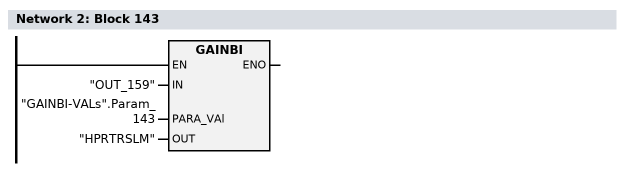
NETWORK
TITLE = Block 143
      CALL  "GAINBI" (
           IN                       := "OUT_159",
           PARA_VAl                 := "GAINBI-VALs".Param_143,
           OUT                      := "HPRTRSLM");
      NOP   0;
END_FUNCTION

FUNCTION "Sheet 23 (RSM)" : VOID	// FC 62
TITLE = Sheet 23 (RSM)
//HP ROTOR STRESS LIMIT (Digital)
AUTHOR : RJ
FAMILY : RSM
VERSION : 0.1
BEGIN
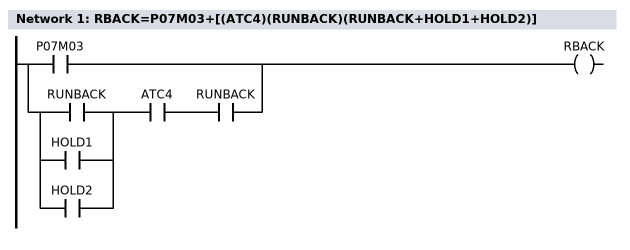
NETWORK
TITLE = RBACK=P07M03+[(ATC4)(RUNBACK)(RUNBACK+HOLD1+HOLD2)]
      O     "P07M03";
      O;
      A(;
      O     "RUNBACK";
      O     "HOLD1";
      O     "HOLD2";
      );
      A     "ATC4";
      A     "RUNBACK";
      =     "RBACK";
NETWORK
TITLE = P01M02=[FF(HILDPB,[NORLDPB+~BR+LDEQDMD])][DVTRUE]
      A(;
      A     "HILDPB";
      S     "HILDRAT";
      A(;
      O     "NORLDPB";
      ON    "BR";
      O     "LDEQDMD";
      );
      R     "HILDRAT";
      A     "HILDRAT";
      );
      A     "Constants_RSM".DVTRUE;
      =     "P01M02";
END_FUNCTION

FUNCTION "Sheet 24 (RSM)" : VOID	// FC 63
TITLE = Sheet 24 (RSM)
//ATC TARGET (Analog)
AUTHOR : RJ
FAMILY : RSM
VERSION : 0.1
BEGIN
NETWORK
TITLE = Blocks X712, X715
      A     "RES1";
      =     L 0.0;
      BLD   103;
      A(;
      A     "HLD1";
      =     L 0.1;
      BLD   103;
      CALL  "XTRANSF" (
           PV_Y                     := "REFDMD",
           CAS_N                    := "OUT_X171",
           FLAG                     := L 0.1,
           PARA_VAl                 := "XTRANSF_VALs".Param_X712,
           OUTPUT                   := "OUT_X712");
      A     BR;
      );
      JNB   _001;
      CALL  "XTRANSF" (
           PV_Y                     := "REFF1",
           CAS_N                    := "OUT_X712",
           FLAG                     := L 0.0,
           PARA_VAl                 := "XTRANSF_VALs".Param_X715,
           OUTPUT                   := "OUT_X715");
_001: NOP   0;
NETWORK
TITLE = Blocks X717, X721
      A     "RES3";
      =     L 0.0;
      BLD   103;
      A(;
      A     "RES2";
      =     L 0.1;
      BLD   103;
      CALL  "XTRANSF" (
           PV_Y                     := "REFF2",
           CAS_N                    := "OUT_X715",
           FLAG                     := L 0.1,
           PARA_VAl                 := "XTRANSF_VALs".Param_X717,
           OUTPUT                   := "DMDTEMP2");
      A     BR;
      );
      JNB   _002;
      CALL  "XTRANSF" (
           PV_Y                     := "REFF3",
           CAS_N                    := "DMDTEMP2",
           FLAG                     := L 0.0,
           PARA_VAl                 := "XTRANSF_VALs".Param_X721,
           OUTPUT                   := "OUT_X721");
_002: NOP   0;
NETWORK
TITLE = Blocks X723, X725
      A     "RES5";
      =     L 0.0;
      BLD   103;
      A(;
      A     "RES4";
      =     L 0.1;
      BLD   103;
      CALL  "XTRANSF" (
           PV_Y                     := "REFF4",
           CAS_N                    := "OUT_X721",
           FLAG                     := L 0.1,
           PARA_VAl                 := "XTRANSF_VALs".Param_X723,
           OUTPUT                   := "OUT_X723");
      A     BR;
      );
      JNB   _003;
      CALL  "XTRANSF" (
           PV_Y                     := "REFF5",
           CAS_N                    := "DMDTEMP3",
           FLAG                     := L 0.0,
           PARA_VAl                 := "XTRANSF_VALs".Param_X725,
           OUTPUT                   := "DMDTEMP3");
_003: NOP   0;
NETWORK
TITLE = Blocks X741, X743
      A     "RBACK";
      =     L 0.0;
      BLD   103;
      A(;
      A     "EXC1";
      =     L 0.1;
      BLD   103;
      CALL  "XTRANSF" (
           PV_Y                     := "Constants_RSM".A40,
           CAS_N                    := "DMDTEMP3",
           FLAG                     := L 0.1,
           PARA_VAl                 := "XTRANSF_VALs".Param_X741,
           OUTPUT                   := "OUT_X741");
      A     BR;
      );
      JNB   _004;
      CALL  "XTRANSF" (
           PV_Y                     := "ATCSPDRF",
           CAS_N                    := "OUT_X741",
           FLAG                     := L 0.0,
           PARA_VAl                 := "XTRANSF_VALs".Param_X743,
           OUTPUT                   := "DEHDMD");
_004: NOP   0;
NETWORK
TITLE = Blocks X701, X707
      A     "DEHDMD1";
      =     L 0.0;
      BLD   103;
      A(;
      A     "P15M13";
      =     L 0.1;
      BLD   103;
      CALL  "XTRANSF" (
           PV_Y                     := "Constants_RSM".A40,
           CAS_N                    := "DEHDMD",
           FLAG                     := L 0.1,
           PARA_VAl                 := "XTRANSF_VALs".Param_X701,
           OUTPUT                   := "OUT_X701");
      A     BR;
      );
      JNB   _005;
      CALL  "XTRANSF" (
           PV_Y                     := "Constants_RSM".A40,
           CAS_N                    := "OUT_X701",
           FLAG                     := L 0.0,
           PARA_VAl                 := "XTRANSF_VALs".Param_X707,
           OUTPUT                   := "OUT_X707");
_005: NOP   0;
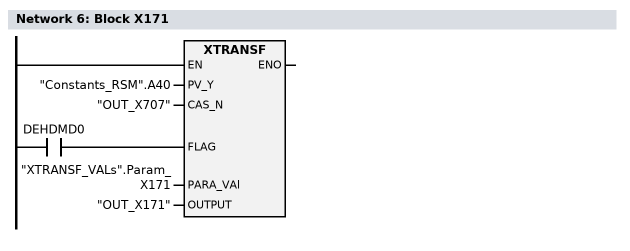
NETWORK
TITLE = Block X171
      A     "DEHDMD0";
      =     L 0.0;
      BLD   103;
      CALL  "XTRANSF" (
           PV_Y                     := "Constants_RSM".A40,
           CAS_N                    := "OUT_X707",
           FLAG                     := L 0.0,
           PARA_VAl                 := "XTRANSF_VALs".Param_X171,
           OUTPUT                   := "OUT_X171");
      NOP   0;
END_FUNCTION

FUNCTION "Sheet 25 (RSM)" : VOID	// FC 64
TITLE = Sheet 25 (RSM)
//TRANSFER DELAY (Digital)
AUTHOR : RJ
FAMILY : RSM
VERSION : 0.1
BEGIN
NETWORK
TITLE = CRSBO4=FF[(AFLAG)(ATC4),(ATC4)(Z871)]
//Z871=ON(CRSBO4)
      A(;
      A     "AFLAG";
      A     "ATC4";
      S     "CRSBO4";
      A     "Z871";
      A     "ATC4";
      R     "CRSBO4";
      A     "CRSBO4";
      );
      =     "CRSBO4";
      A     "CRSBO4";
      L     "RSMTime_VALs".T1ON;
      SD    T 1;
      NOP   0;
      NOP   0;
      NOP   0;
      A     T 1;
      =     "Z871";
END_FUNCTION

FUNCTION "Sheet 26 (RSM)" : VOID	// FC 65
TITLE = Sheet 26 (RSM)
//LADDERS 35, 128, RESONANCE RANGE LOGIC (Digital)
AUTHOR : RJ
FAMILY : RSM
VERSION : 0.1
BEGIN
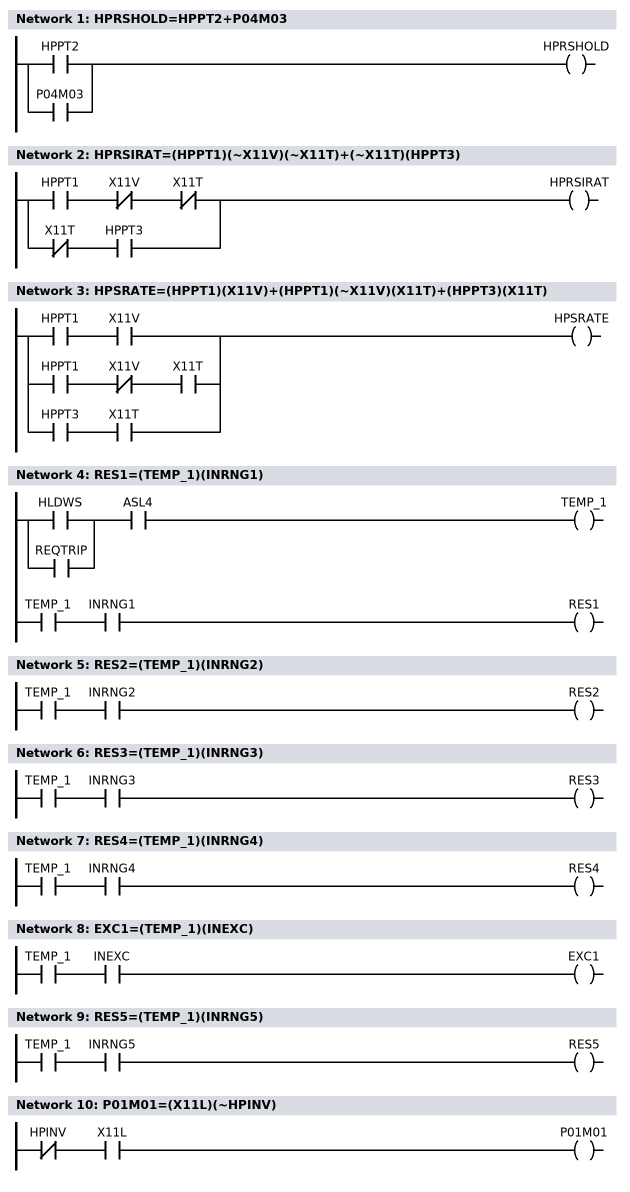
NETWORK
TITLE = HPRSHOLD=HPPT2+P04M03
      O     "HPPT2";
      O     "P04M03";
      =     "HPRSHOLD";
NETWORK
TITLE = HPRSIRAT=(HPPT1)(~X11V)(~X11T)+(~X11T)(HPPT3)
      A     "HPPT1";
      AN    "X11V";
      AN    "X11T";
      O;
      AN    "X11T";
      A     "HPPT3";
      =     "HPRSIRAT";
NETWORK
TITLE = HPSRATE=(HPPT1)(X11V)+(HPPT1)(~X11V)(X11T)+(HPPT3)(X11T)
      A     "HPPT1";
      A     "X11V";
      O;
      A     "HPPT1";
      AN    "X11V";
      A     "X11T";
      O;
      A     "HPPT3";
      A     "X11T";
      =     "HPSRATE";
NETWORK
TITLE = RES1=(TEMP_1)(INRNG1)
//TEMP_1=(ASL4)(HLDWS+REQTRIP)
      A(;
      O     "HLDWS";
      O     "REQTRIP";
      );
      A     "ASL4";
      =     "TEMP_1";
      A     "TEMP_1";
      A     "INRNG1";
      =     "RES1";
NETWORK
TITLE = RES2=(TEMP_1)(INRNG2)
      A     "TEMP_1";
      A     "INRNG2";
      =     "RES2";
NETWORK
TITLE = RES3=(TEMP_1)(INRNG3)
      A     "TEMP_1";
      A     "INRNG3";
      =     "RES3";
NETWORK
TITLE = RES4=(TEMP_1)(INRNG4)
      A     "TEMP_1";
      A     "INRNG4";
      =     "RES4";
NETWORK
TITLE = EXC1=(TEMP_1)(INEXC)
      A     "TEMP_1";
      A     "INEXC";
      =     "EXC1";
NETWORK
TITLE = RES5=(TEMP_1)(INRNG5)
      A     "TEMP_1";
      A     "INRNG5";
      =     "RES5";
NETWORK
TITLE = P01M01=(X11L)(~HPINV)
      AN    "HPINV";
      A     "X11L";
      =     "P01M01";
END_FUNCTION

FUNCTION "Sheet 28 (RSM)" : VOID	// FC 66
TITLE = Sheet 28 (RSM)
//LADDERS 22, 500, 600, DIGITAL POINTERS TMAX & TWC LOGIC (Digital)
AUTHOR : RJ
FAMILY : RSM
VERSION : 0.1
BEGIN
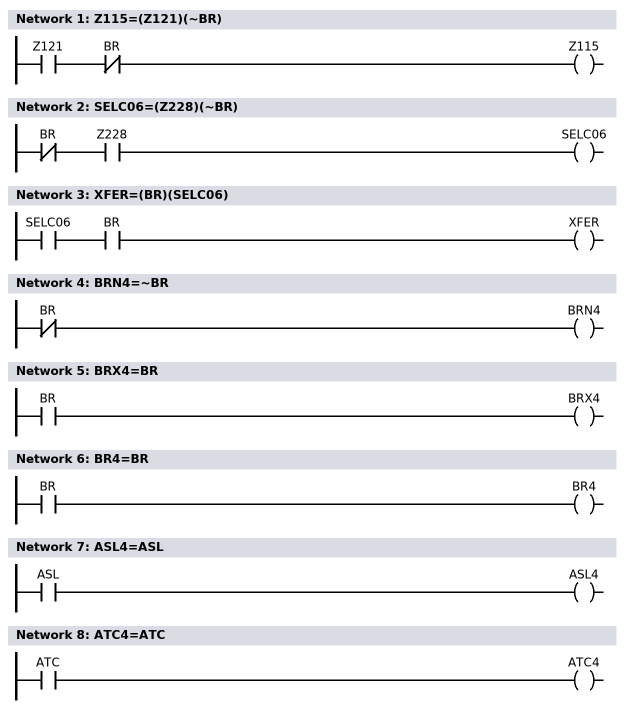
NETWORK
TITLE = Z115=(Z121)(~BR)
      A     "Z121";
      AN    "BR";
      =     "Z115";
NETWORK
TITLE = SELC06=(Z228)(~BR)
      AN    "BR";
      A     "Z228";
      =     "SELC06";
NETWORK
TITLE = XFER=(BR)(SELC06)
      A     "SELC06";
      A     "BR";
      =     "XFER";
NETWORK
TITLE = BRN4=~BR
      AN    "BR";
      =     "BRN4";
NETWORK
TITLE = BRX4=BR
      A     "BR";
      =     "BRX4";
NETWORK
TITLE = BR4=BR
      A     "BR";
      =     "BR4";
NETWORK
TITLE = ASL4=ASL
      A     "ASL";
      =     "ASL4";
NETWORK
TITLE = ATC4=ATC
      A     "ATC";
      =     "ATC4";
END_FUNCTION

FUNCTION "Sheet 29 (RSM)" : VOID	// FC 67
TITLE = Sheet 29 (RSM)
//LADDERS 29, 31, 500, FIRST STAGE STM > 75 *C (Digital)
AUTHOR : RJ
FAMILY : RSM
VERSION : 0.1
BEGIN
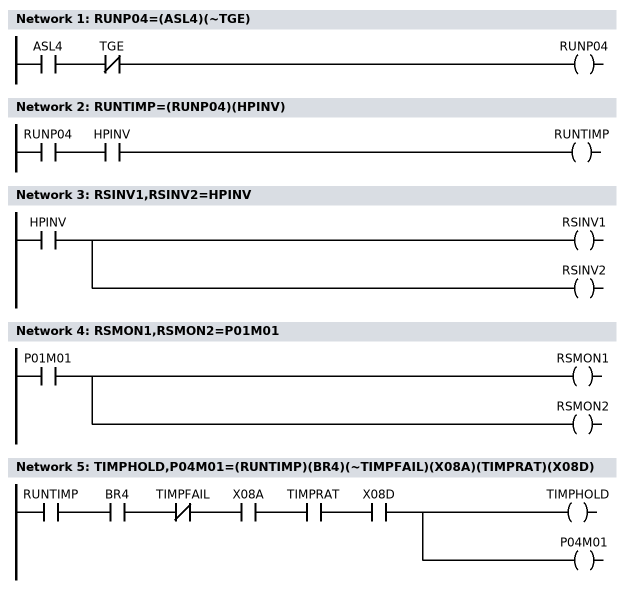
NETWORK
TITLE = RUNP04=(ASL4)(~TGE)
      A     "ASL4";
      AN    "TGE";
      =     "RUNP04";
NETWORK
TITLE = RUNTIMP=(RUNP04)(HPINV)
      A     "RUNP04";
      A     "HPINV";
      =     "RUNTIMP";
NETWORK
TITLE = RSINV1,RSINV2=HPINV
      A     "HPINV";
      =     "RSINV1";
      =     "RSINV2";
NETWORK
TITLE = RSMON1,RSMON2=P01M01
      A     "P01M01";
      =     "RSMON1";
      =     "RSMON2";
NETWORK
TITLE = TIMPHOLD,P04M01=(RUNTIMP)(BR4)(~TIMPFAIL)(X08A)(TIMPRAT)(X08D)
      A     "RUNTIMP";
      A     "BR4";
      AN    "TIMPFAIL";
      A     "X08A";
      A     "TIMPRAT";
      A     "X08D";
      =     "TIMPHOLD";
      =     "P04M01";
END_FUNCTION

FUNCTION "Sheet 27 (RSM)" : VOID	// FC 68
TITLE = Sheet 27 (RSM)
//LADDERS 43, 129, RTSHOLD (Digital)
AUTHOR : RJ
FAMILY : RSM
VERSION : 0.1
BEGIN
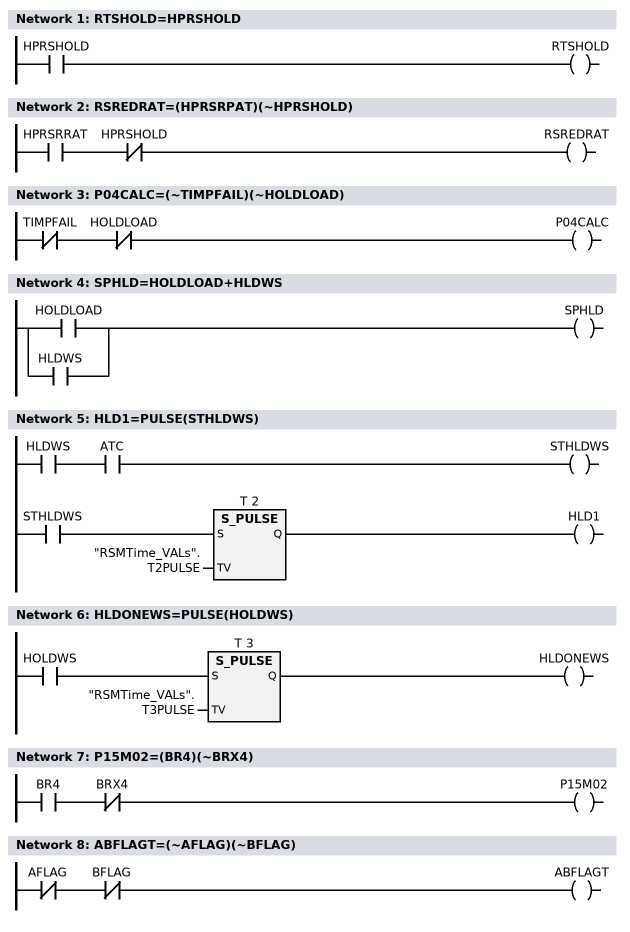
NETWORK
TITLE = RTSHOLD=HPRSHOLD
      A     "HPRSHOLD";
      =     "RTSHOLD";
NETWORK
TITLE = RSREDRAT=(HPRSRPAT)(~HPRSHOLD)
      A     "HPRSRRAT";
      AN    "HPRSHOLD";
      =     "RSREDRAT";
NETWORK
TITLE = P04CALC=(~TIMPFAIL)(~HOLDLOAD)
      AN    "TIMPFAIL";
      AN    "HOLDLOAD";
      =     "P04CALC";
NETWORK
TITLE = SPHLD=HOLDLOAD+HLDWS
      O     "HOLDLOAD";
      O     "HLDWS";
      =     "SPHLD";
NETWORK
TITLE = HLD1=PULSE(STHLDWS)
//STHLDWS=(HLDWS)(ATC)
      A     "HLDWS";
      A     "ATC";
      =     "STHLDWS";
      A     "STHLDWS";
      L     "RSMTime_VALs".T2PULSE;
      SP    T 2;
      NOP   0;
      NOP   0;
      NOP   0;
      A     T 2;
      =     "HLD1";
NETWORK
TITLE = HLDONEWS=PULSE(HOLDWS)
      A     "HOLDWS";
      L     "RSMTime_VALs".T3PULSE;
      SP    T 3;
      NOP   0;
      NOP   0;
      NOP   0;
      A     T 3;
      =     "HLDONEWS";
NETWORK
TITLE = P15M02=(BR4)(~BRX4)
      A     "BR4";
      AN    "BRX4";
      =     "P15M02";
NETWORK
TITLE = ABFLAGT=(~AFLAG)(~BFLAG)
      AN    "AFLAG";
      AN    "BFLAG";
      =     "ABFLAGT";
END_FUNCTION

FUNCTION "Sheet 30 (RSM)" : VOID	// FC 69
TITLE = Sheet 30 (RSM)
//LADDER 126, SYNC LOGIC & OVERRIDE (Digital)
AUTHOR : RJ
FAMILY : RSM
VERSION : 0.1
BEGIN
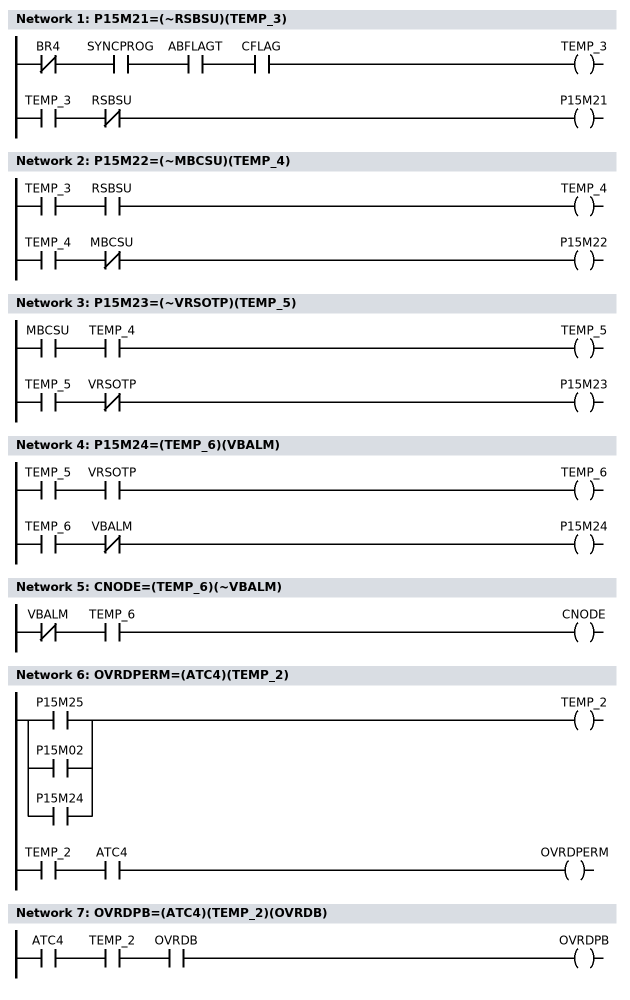
NETWORK
TITLE = P15M21=(~RSBSU)(TEMP_3)
//TEMP_3=(~BR4)(SYNCPROG)(ABFLAGT)(CFLAG)
      AN    "BR4";
      A     "SYNCPROG";
      A     "ABFLAGT";
      A     "CFLAG";
      =     "TEMP_3";
      A     "TEMP_3";
      AN    "RSBSU";
      =     "P15M21";
NETWORK
TITLE = P15M22=(~MBCSU)(TEMP_4)
//TEMP_4=(TEMP_3)(RSBSU)
      A     "TEMP_3";
      A     "RSBSU";
      =     "TEMP_4";
      A     "TEMP_4";
      AN    "MBCSU";
      =     "P15M22";
NETWORK
TITLE = P15M23=(~VRSOTP)(TEMP_5)
//TEMP_5=(MBCSU)(TEMP_4)
      A     "MBCSU";
      A     "TEMP_4";
      =     "TEMP_5";
      A     "TEMP_5";
      AN    "VRSOTP";
      =     "P15M23";
NETWORK
TITLE = P15M24=(TEMP_6)(VBALM)
//TEMP_6=(TEMP_5)(VRSOTP)
      A     "TEMP_5";
      A     "VRSOTP";
      =     "TEMP_6";
      A     "TEMP_6";
      AN    "VBALM";
      =     "P15M24";
NETWORK
TITLE = CNODE=(TEMP_6)(~VBALM)
      AN    "VBALM";
      A     "TEMP_6";
      =     "CNODE";
NETWORK
TITLE = OVRDPERM=(ATC4)(TEMP_2)
//TEMP_2=P15M25+P15M06+P15M24
      A(;
      O     "P15M25";
      O     "P15M02";
      O     "P15M24";
      );
      =     "TEMP_2";
      A     "TEMP_2";
      A     "ATC4";
      =     "OVRDPERM";
NETWORK
TITLE = OVRDPB=(ATC4)(TEMP_2)(OVRDB)
      A     "ATC4";
      A     "TEMP_2";
      A     "OVRDB";
      =     "OVRDPB";
END_FUNCTION

FUNCTION "Sheet 31 (RSM)" : VOID	// FC 70
TITLE = Sheet 31 (RSM)
//LADDER 33, ANTIC HP STRESS > LIMIT (Digital)
AUTHOR : RJ
FAMILY : RSM
VERSION : 0.1
BEGIN
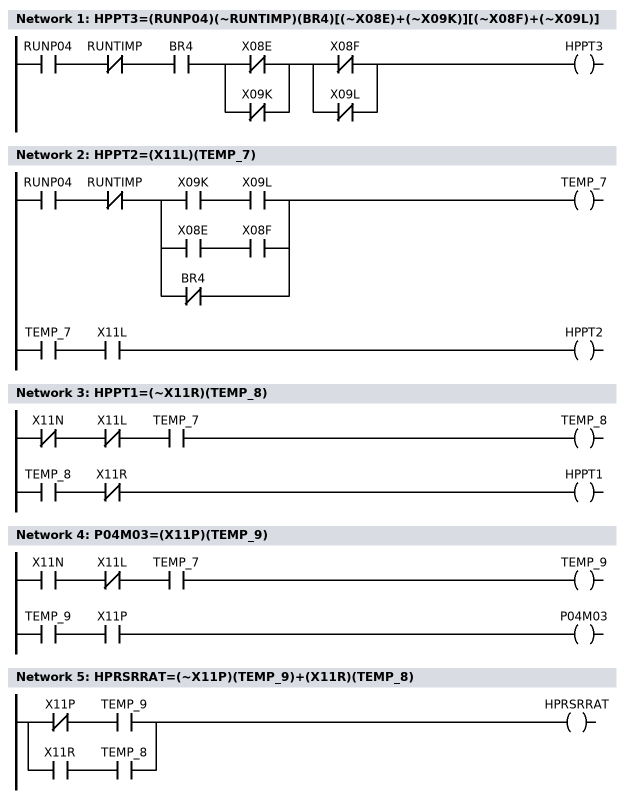
NETWORK
TITLE = HPPT3=(RUNP04)(~RUNTIMP)(BR4)[(~X08E)+(~X09K)][(~X08F)+(~X09L)]
      A     "RUNP04";
      AN    "RUNTIMP";
      A     "BR4";
      A(;
      ON    "X08E";
      ON    "X09K";
      );
      A(;
      ON    "X08F";
      ON    "X09L";
      );
      =     "HPPT3";
NETWORK
TITLE = HPPT2=(X11L)(TEMP_7)
//TEMP_7=(RUNP04)(~RUNTIMP)[(X09K)(X09L)+(X08E)(X08F)+(~BR4)]
      A     "RUNP04";
      AN    "RUNTIMP";
      A(;
      A     "X09K";
      A     "X09L";
      O;
      A     "X08E";
      A     "X08F";
      ON    "BR4";
      );
      =     "TEMP_7";
      A     "TEMP_7";
      A     "X11L";
      =     "HPPT2";
NETWORK
TITLE = HPPT1=(~X11R)(TEMP_8)
//TEMP_8=(~X11N)(~X11L)(TEMP_7)
      AN    "X11N";
      AN    "X11L";
      A     "TEMP_7";
      =     "TEMP_8";
      A     "TEMP_8";
      AN    "X11R";
      =     "HPPT1";
NETWORK
TITLE = P04M03=(X11P)(TEMP_9)
//TEMP_9=(X11N)(~X11L)(TEMP_7)
      A     "X11N";
      AN    "X11L";
      A     "TEMP_7";
      =     "TEMP_9";
      A     "TEMP_9";
      A     "X11P";
      =     "P04M03";
NETWORK
TITLE = HPRSRRAT=(~X11P)(TEMP_9)+(X11R)(TEMP_8)
      AN    "X11P";
      A     "TEMP_9";
      O;
      A     "X11R";
      A     "TEMP_8";
      =     "HPRSRRAT";
END_FUNCTION

FUNCTION "Sheet 32 (RSM)" : VOID	// FC 71
TITLE = Sheet 32 (RSM)
//LADDERS 37, 125, 130, SYNC LOGIC & OVERRIDE (Digital)
AUTHOR : RJ
FAMILY : RSM
VERSION : 0.1
BEGIN
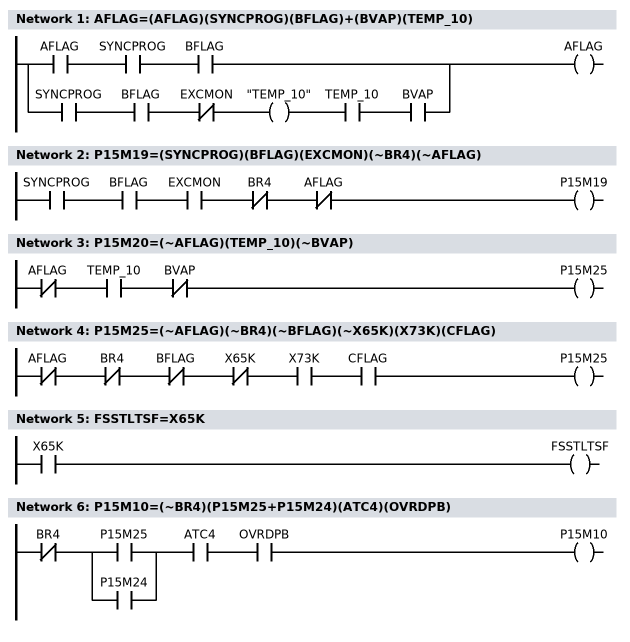
NETWORK
TITLE = AFLAG=(AFLAG)(SYNCPROG)(BFLAG)+(BVAP)(TEMP_10)
//TEMP_10=(SYNCPROG)(BFLAG)(~EXCMON)
      A     "AFLAG";
      A     "SYNCPROG";
      A     "BFLAG";
      O(;
      A     "SYNCPROG";
      A     "BFLAG";
      AN    "EXCMON";
      =     "TEMP_10";
      A     "TEMP_10";
      A     "BVAP";
      );
      =     "AFLAG";
NETWORK
TITLE = P15M19=(SYNCPROG)(BFLAG)(EXCMON)(~BR4)(~AFLAG)
      A     "SYNCPROG";
      A     "BFLAG";
      A     "EXCMON";
      AN    "BR4";
      AN    "AFLAG";
      =     "P15M19";
NETWORK
TITLE = P15M20=(~AFLAG)(TEMP_10)(~BVAP)
      AN    "AFLAG";
      A     "TEMP_10";
      AN    "BVAP";
      =     "P15M25";
NETWORK
TITLE = P15M25=(~AFLAG)(~BR4)(~BFLAG)(~X65K)(X73K)(CFLAG)
      AN    "AFLAG";
      AN    "BR4";
      AN    "BFLAG";
      AN    "X65K";
      A     "X73K";
      A     "CFLAG";
      =     "P15M25";
NETWORK
TITLE = FSSTLTSF=X65K
      A     "X65K";
      =     "FSSTLTSF";
NETWORK
TITLE = P15M10=(~BR4)(P15M25+P15M24)(ATC4)(OVRDPB)
      AN    "BR4";
      A(;
      O     "P15M25";
      O     "P15M24";
      );
      A     "ATC4";
      A     "OVRDPB";
      =     "P15M10";
END_FUNCTION

FUNCTION "Sheet 33 (RSM)" : VOID	// FC 72
TITLE = Sheet 33 (RSM)
//LADDER 124, 127, SYNC LOGIC & TVGVINIT (Digital)
AUTHOR : RJ
FAMILY : RSM
VERSION : 0.1
BEGIN
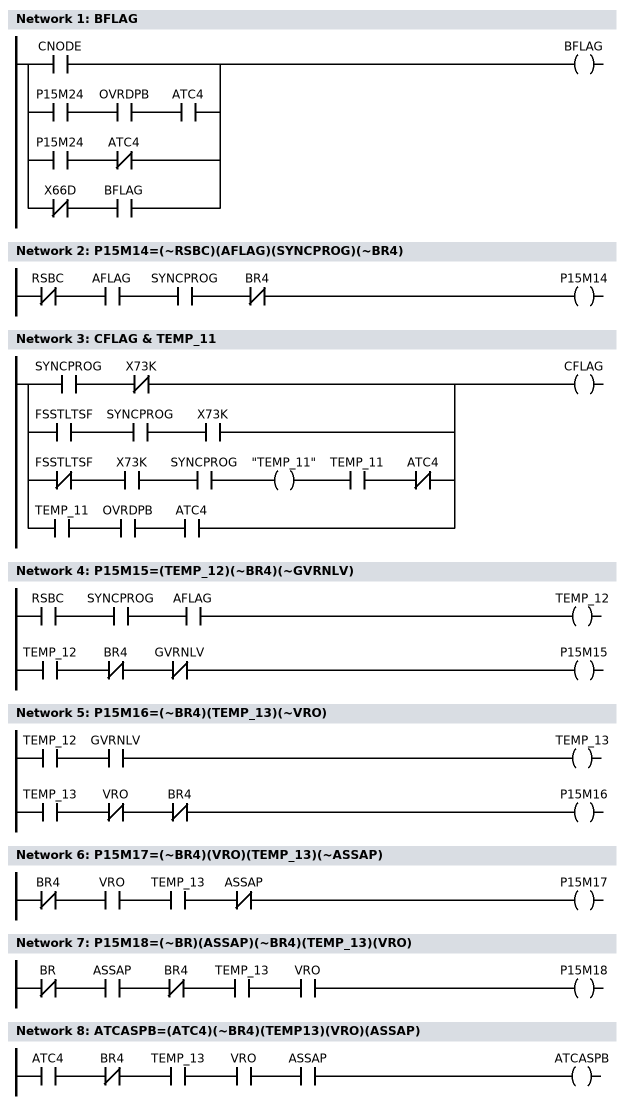
NETWORK
TITLE = BFLAG
//BFLAG=CNODE+(P15M24)(OVRDPB)(ATC4)+(P15M24)(~ATC4)+(~X66D)(BFLAG)
      O     "CNODE";
      O;
      A     "P15M24";
      A     "OVRDPB";
      A     "ATC4";
      O;
      A     "P15M24";
      AN    "ATC4";
      O;
      AN    "X66D";
      A     "BFLAG";
      =     "BFLAG";
NETWORK
TITLE = P15M14=(~RSBC)(AFLAG)(SYNCPROG)(~BR4)
      AN    "RSBC";
      A     "AFLAG";
      A     "SYNCPROG";
      AN    "BR4";
      =     "P15M14";
NETWORK
TITLE = CFLAG & TEMP_11
//CFLAG=(SYNCPROG)(~X73K)+(FSSTLTSF)(SYNCPROG)(X73K)+(~ATC4)(TEMP_11)+(TEMP_11)
//(OVRDPB)(ATC4)
//
//TEMP_11=(~FSSTLTSF)(X73K)(SYNCPROG)
//
      A     "SYNCPROG";
      AN    "X73K";
      O(;
      A     "FSSTLTSF";
      A     "SYNCPROG";
      A     "X73K";
      );
      O(;
      AN    "FSSTLTSF";
      A     "X73K";
      A     "SYNCPROG";
      =     "TEMP_11";
      A     "TEMP_11";
      AN    "ATC4";
      );
      O;
      A     "TEMP_11";
      A     "OVRDPB";
      A     "ATC4";
      =     "CFLAG";
NETWORK
TITLE = P15M15=(TEMP_12)(~BR4)(~GVRNLV)
//TEMP_12=(RSBC)(SYNCPROG)(AFLAG)
      A     "RSBC";
      A     "SYNCPROG";
      A     "AFLAG";
      =     "TEMP_12";
      A     "TEMP_12";
      AN    "BR4";
      AN    "GVRNLV";
      =     "P15M15";
NETWORK
TITLE = P15M16=(~BR4)(TEMP_13)(~VRO)
//TEMP_13=(TEMP_12)(GVRNLV)
      A     "TEMP_12";
      A     "GVRNLV";
      =     "TEMP_13";
      A     "TEMP_13";
      AN    "VRO";
      AN    "BR4";
      =     "P15M16";
NETWORK
TITLE = P15M17=(~BR4)(VRO)(TEMP_13)(~ASSAP)
      AN    "BR4";
      A     "VRO";
      A     "TEMP_13";
      AN    "ASSAP";
      =     "P15M17";
NETWORK
TITLE = P15M18=(~BR)(ASSAP)(~BR4)(TEMP_13)(VRO)
      AN    "BR";
      A     "ASSAP";
      AN    "BR4";
      A     "TEMP_13";
      A     "VRO";
      =     "P15M18";
NETWORK
TITLE = ATCASPB=(ATC4)(~BR4)(TEMP13)(VRO)(ASSAP)
      A     "ATC4";
      AN    "BR4";
      A     "TEMP_13";
      A     "VRO";
      A     "ASSAP";
      =     "ATCASPB";
END_FUNCTION

FUNCTION "Sheet 34 (RSM)" : VOID	// FC 73
TITLE = Sheet 34 (RSM)
//LADDERS 122, 123, 135, SET SPEED PLATEAU (Digital)
AUTHOR : RJ
FAMILY : RSM
VERSION : 0.1
BEGIN
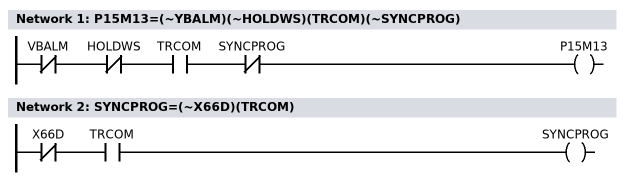
NETWORK
TITLE = P15M13=(~YBALM)(~HOLDWS)(TRCOM)(~SYNCPROG)
      AN    "VBALM";
      AN    "HOLDWS";
      A     "TRCOM";
      AN    "SYNCPROG";
      =     "P15M13";
NETWORK
TITLE = SYNCPROG=(~X66D)(TRCOM)
      AN    "X66D";
      A     "TRCOM";
      =     "SYNCPROG";
END_FUNCTION

FUNCTION "Sheet 35 (RSM)" : VOID	// FC 74
TITLE = Sheet 35 (RSM)
//LADDER 120, 121, P15 ALARMS ESTIMATE ROLL TIME LOGIC & ATC VPL (Digital)
AUTHOR : RJ
FAMILY : RSM
VERSION : 0.1
BEGIN
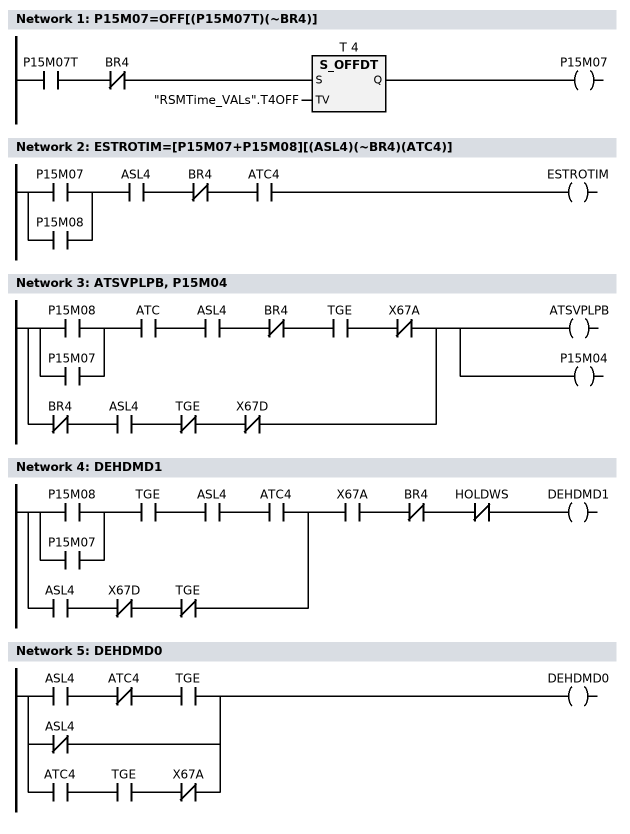
NETWORK
TITLE = P15M07=OFF[(P15M07T)(~BR4)]
      A     "P15M07T";
      AN    "BR4";
      L     "RSMTime_VALs".T4OFF;
      SF    T 4;
      NOP   0;
      NOP   0;
      NOP   0;
      A     T 4;
      =     "P15M07";
NETWORK
TITLE = ESTROTIM=[P15M07+P15M08][(ASL4)(~BR4)(ATC4)]
      A(;
      O     "P15M07";
      O     "P15M08";
      );
      A     "ASL4";
      AN    "BR4";
      A     "ATC4";
      =     "ESTROTIM";
NETWORK
TITLE = ATSVPLPB, P15M04
//ATSVPLPB,P15M04=[(P15M08+P15M07)(ATC)(ASL4)(~BR4)(TGE)(~X67A)]+[(~BR4)(ASL4)
//(~TGE)(~X67D)]
      A(;
      O     "P15M08";
      O     "P15M07";
      );
      A     "ATC";
      A     "ASL4";
      AN    "BR4";
      A     "TGE";
      AN    "X67A";
      O;
      AN    "BR4";
      A     "ASL4";
      AN    "TGE";
      AN    "X67D";
      =     "ATSVPLPB";
      =     "P15M04";
NETWORK
TITLE = DEHDMD1
//DEHDMD1=[{(P15M08+P15M07)(TGE)(ASL4)(ATC4)}+{(ASL4)(~X67D)(~TGE)}][X67A][~BR4]
//[~HOLDWS]
      A(;
      A(;
      O     "P15M08";
      O     "P15M07";
      );
      A     "TGE";
      A     "ASL4";
      A     "ATC4";
      O;
      A     "ASL4";
      AN    "X67D";
      AN    "TGE";
      );
      A     "X67A";
      AN    "BR4";
      AN    "HOLDWS";
      =     "DEHDMD1";
NETWORK
TITLE = DEHDMD0
//DEHDMD0=[(ASL4)(~ATC4)(TGE)]+[~ASL4]+[(ASL4)(TGE)(~X67A)]
      A     "ASL4";
      AN    "ATC4";
      A     "TGE";
      ON    "ASL4";
      O;
      A     "ATC4";
      A     "TGE";
      AN    "X67A";
      =     "DEHDMD0";
END_FUNCTION

FUNCTION "Sheet 36 (RSM)" : VOID	// FC 75
TITLE = Sheet 36 (RSM)
//LADDER 41, 119, P15 ALARMS (Digital)
AUTHOR : RJ
FAMILY : RSM
VERSION : 0.1
BEGIN
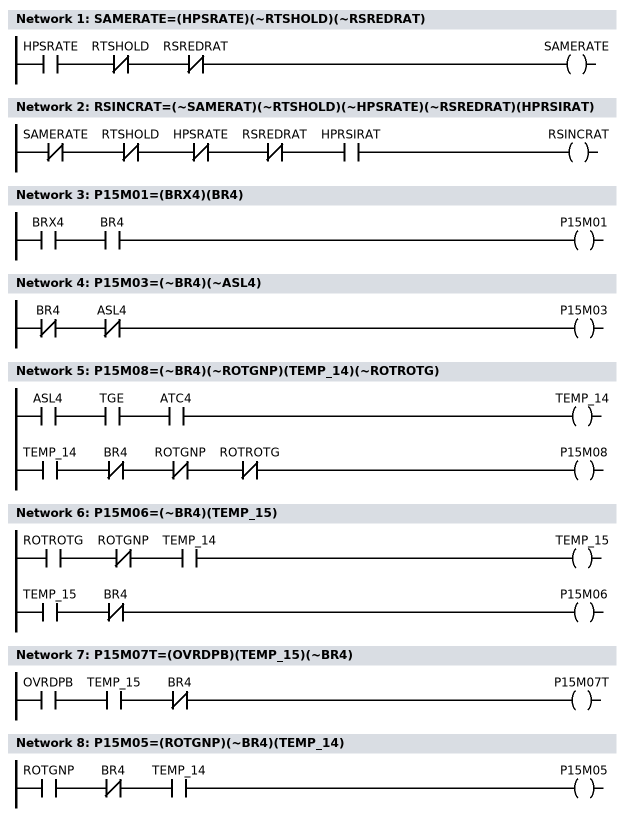
NETWORK
TITLE = SAMERATE=(HPSRATE)(~RTSHOLD)(~RSREDRAT)
      A     "HPSRATE";
      AN    "RTSHOLD";
      AN    "RSREDRAT";
      =     "SAMERATE";
NETWORK
TITLE = RSINCRAT=(~SAMERAT)(~RTSHOLD)(~HPSRATE)(~RSREDRAT)(HPRSIRAT)
      AN    "SAMERATE";
      AN    "RTSHOLD";
      AN    "HPSRATE";
      AN    "RSREDRAT";
      A     "HPRSIRAT";
      =     "RSINCRAT";
NETWORK
TITLE = P15M01=(BRX4)(BR4)
      A     "BRX4";
      A     "BR4";
      =     "P15M01";
NETWORK
TITLE = P15M03=(~BR4)(~ASL4)
      AN    "BR4";
      AN    "ASL4";
      =     "P15M03";
NETWORK
TITLE = P15M08=(~BR4)(~ROTGNP)(TEMP_14)(~ROTROTG)
//TEMP_14=(ASL4)(TGE)(ATC4)
      A     "ASL4";
      A     "TGE";
      A     "ATC4";
      =     "TEMP_14";
      A     "TEMP_14";
      AN    "BR4";
      AN    "ROTGNP";
      AN    "ROTROTG";
      =     "P15M08";
NETWORK
TITLE = P15M06=(~BR4)(TEMP_15)
//TEMP_15=(ROTROTG)(~ROTGNP)(TEMP_14)
      A     "ROTROTG";
      AN    "ROTGNP";
      A     "TEMP_14";
      =     "TEMP_15";
      A     "TEMP_15";
      AN    "BR4";
      =     "P15M06";
NETWORK
TITLE = P15M07T=(OVRDPB)(TEMP_15)(~BR4)
      A     "OVRDPB";
      A     "TEMP_15";
      AN    "BR4";
      =     "P15M07T";
NETWORK
TITLE = P15M05=(ROTGNP)(~BR4)(TEMP_14)
      A     "ROTGNP";
      AN    "BR4";
      A     "TEMP_14";
      =     "P15M05";
END_FUNCTION

FUNCTION "Sheet 37 (RSM)" : VOID	// FC 76
TITLE = Sheet 37 (RSM)
//GENERATOR AND EXCITOR TEMPERATURES (Analog)
AUTHOR : RJ
FAMILY : RSM
VERSION : 0.1
BEGIN
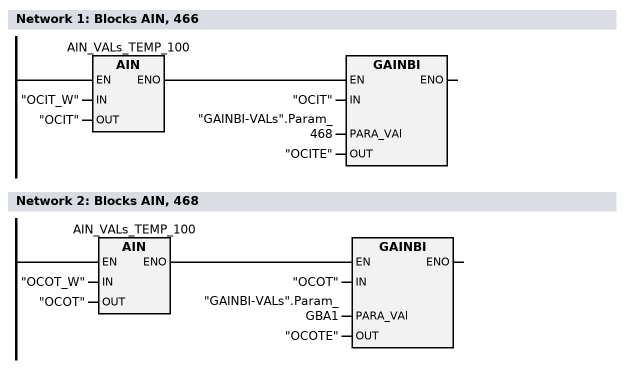
NETWORK
TITLE = Blocks AIN, 466
      A(;
      CALL  "AIN" , "AIN_VALs_TEMP_100" (
           IN                       := "OCIT_W",
           OUT                      := "OCIT");
      A     BR;
      );
      JNB   _001;
      CALL  "GAINBI" (
           IN                       := "OCIT",
           PARA_VAl                 := "GAINBI-VALs".Param_468,
           OUT                      := "OCITE");
_001: NOP   0;
NETWORK
TITLE = Blocks AIN, 468
      A(;
      CALL  "AIN" , "AIN_VALs_TEMP_100" (
           IN                       := "OCOT_W",
           OUT                      := "OCOT");
      A     BR;
      );
      JNB   _002;
      CALL  "GAINBI" (
           IN                       := "OCOT",
           PARA_VAl                 := "GAINBI-VALs".Param_GBA1,
           OUT                      := "OCOTE");
_002: NOP   0;
END_FUNCTION

FUNCTION "Sheet 2 (ATC)" : VOID	// FC 77
TITLE = Sheet 2 (ATC)
//LADDER 500, SENSOR FAIL (Digital)
AUTHOR : RJ
FAMILY : ATC
VERSION : 0.1
BEGIN
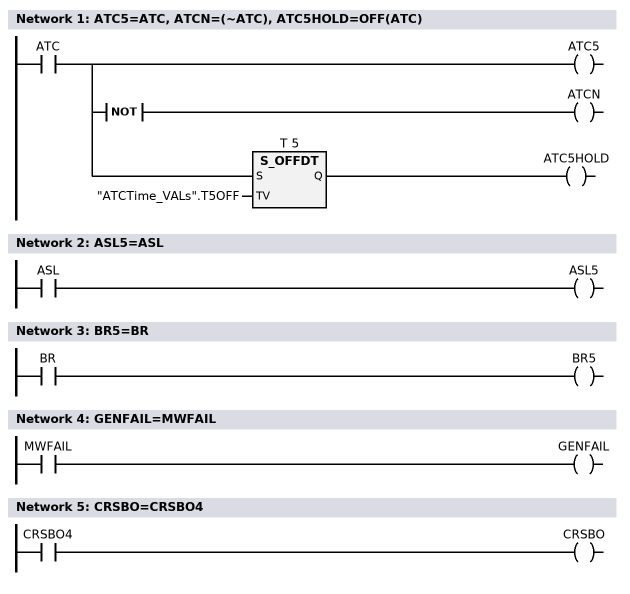
NETWORK
TITLE = ATC5=ATC, ATCN=(~ATC), ATC5HOLD=OFF(ATC)
      A     "ATC";
      =     L 0.0;
      A     L 0.0;
      BLD   102;
      =     "ATC5";
      A     L 0.0;
      NOT;
      =     "ATCN";
      A     L 0.0;
      L     "ATCTime_VALs".T5OFF;
      SF    T 5;
      NOP   0;
      NOP   0;
      NOP   0;
      A     T 5;
      =     "ATC5HOLD";
NETWORK
TITLE = ASL5=ASL
      A     "ASL";
      =     "ASL5";
NETWORK
TITLE = BR5=BR
      A     "BR";
      =     "BR5";
NETWORK
TITLE = GENFAIL=MWFAIL
      A     "MWFAIL";
      =     "GENFAIL";
NETWORK
TITLE = CRSBO=CRSBO4
      A     "CRSBO4";
      =     "CRSBO";
END_FUNCTION

FUNCTION "Sheet 3 (ATC)" : VOID	// FC 78
TITLE = Sheet 3 (ATC)
//SENSOR FAIL (Digital)
AUTHOR : RJ
FAMILY : ATC
VERSION : 0.1
BEGIN
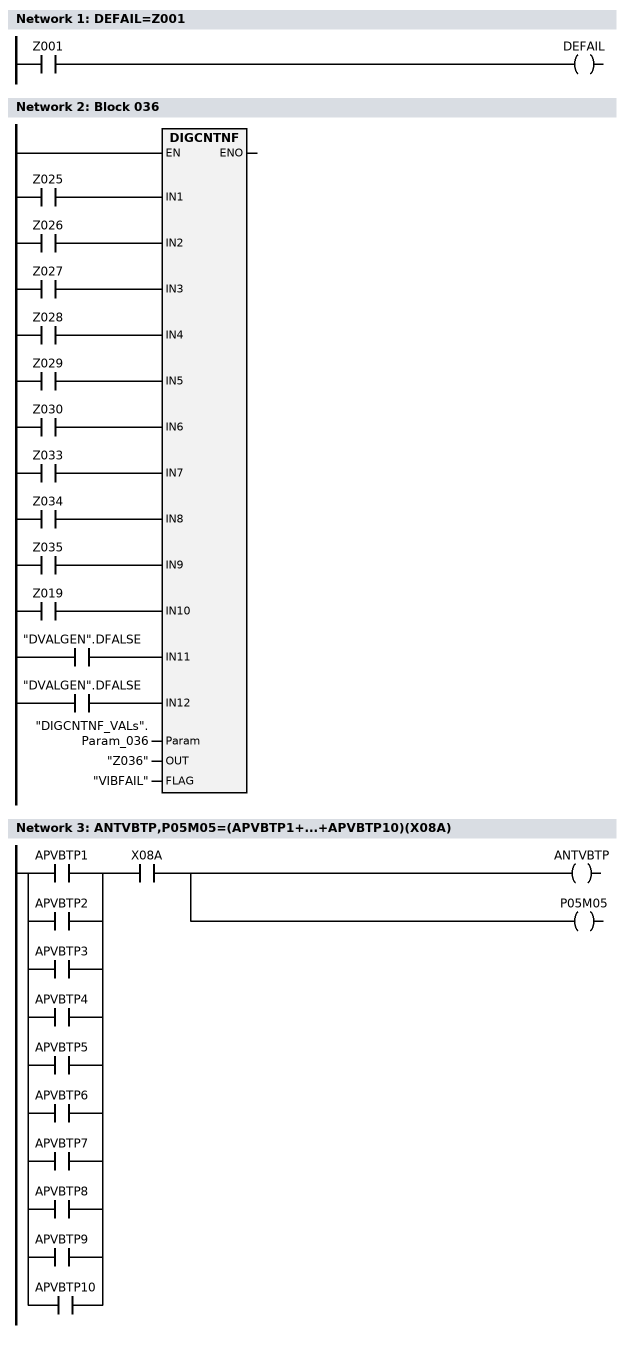
NETWORK
TITLE = DEFAIL=Z001
      A     "Z001";
      =     "DEFAIL";
NETWORK
TITLE = Block 036
      A     "Z025";
      =     L 0.0;
      BLD   103;
      A     "Z026";
      =     L 0.1;
      BLD   103;
      A     "Z027";
      =     L 0.2;
      BLD   103;
      A     "Z028";
      =     L 0.3;
      BLD   103;
      A     "Z029";
      =     L 0.4;
      BLD   103;
      A     "Z030";
      =     L 0.5;
      BLD   103;
      A     "Z033";
      =     L 0.6;
      BLD   103;
      A     "Z034";
      =     L 0.7;
      BLD   103;
      A     "Z035";
      =     L 1.0;
      BLD   103;
      A     "Z019";
      =     L 1.1;
      BLD   103;
      A     "DVALGEN".DFALSE;
      =     L 1.2;
      BLD   103;
      A     "DVALGEN".DFALSE;
      =     L 1.3;
      BLD   103;
      CALL  "DIGCNTNF" (
           IN1                      := L 0.0,
           IN2                      := L 0.1,
           IN3                      := L 0.2,
           IN4                      := L 0.3,
           IN5                      := L 0.4,
           IN6                      := L 0.5,
           IN7                      := L 0.6,
           IN8                      := L 0.7,
           IN9                      := L 1.0,
           IN10                     := L 1.1,
           IN11                     := L 1.2,
           IN12                     := L 1.3,
           Param                    := "DIGCNTNF_VALs".Param_036,
           OUT                      := "Z036",
           FLAG                     := "VIBFAIL");
      NOP   0;
NETWORK
TITLE = ANTVBTP,P05M05=(APVBTP1+...+APVBTP10)(X08A)
      A(;
      O     "APVBTP1";
      O     "APVBTP2";
      O     "APVBTP3";
      O     "APVBTP4";
      O     "APVBTP5";
      O     "APVBTP6";
      O     "APVBTP7";
      O     "APVBTP8";
      O     "APVBTP9";
      O     "APVBTP10";
      );
      A     "X08A";
      =     "ANTVBTP";
      =     "P05M05";
END_FUNCTION

FUNCTION "DIGCNTNF" : VOID	// FC 79
AUTHOR : RJ
VERSION : 0.0
VAR_INPUT
  IN1 : BOOL ;
  IN2 : BOOL ;
  IN3 : BOOL ;
  IN4 : BOOL ;
  IN5 : BOOL ;
  IN6 : BOOL ;
  IN7 : BOOL ;
  IN8 : BOOL ;
  IN9 : BOOL ;
  IN10 : BOOL ;
  IN11 : BOOL ;
  IN12 : BOOL ;
  Param : STRUCT
   N : INT ;
   M : INT ;
  END_STRUCT ;
END_VAR
VAR_OUTPUT
  OUT : INT ;
  FLAG : BOOL ;
END_VAR
VAR_TEMP
  N : INT ;
  M : INT ;
END_VAR
BEGIN
// body was compiled from an SCL source; compiled code not shown
END_FUNCTION

FUNCTION "Sheet 4 (ATC)" : VOID	// FC 81
TITLE = Sheet 4 (ATC)
//LADDERS 1, 3 (Digital)
AUTHOR : RJ
FAMILY : ATC
VERSION : 0.1
BEGIN
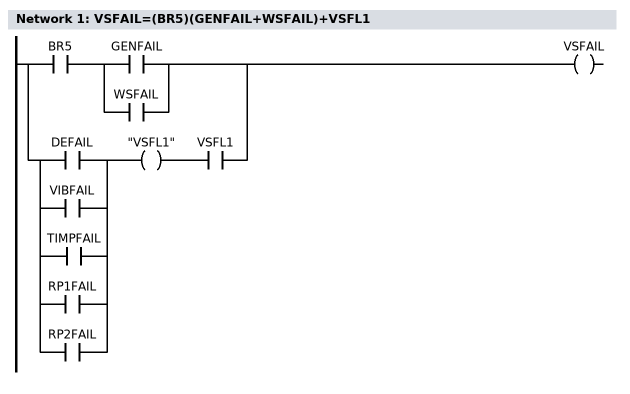
NETWORK
TITLE = VSFAIL=(BR5)(GENFAIL+WSFAIL)+VSFL1
//VSFL1=DEFAIL+VIBFAIL+TIMPFAIL+RP1FAIL+RP2FAIL
      A     "BR5";
      A(;
      O     "GENFAIL";
      O     "WSFAIL";
      );
      O(;
      A(;
      O     "DEFAIL";
      O     "VIBFAIL";
      O     "TIMPFAIL";
      O     "RP1FAIL";
      O     "RP2FAIL";
      );
      =     "VSFL1";
      A     "VSFL1";
      );
      =     "VSFAIL";
END_FUNCTION

FUNCTION "Sheet 5 (ATC)" : VOID	// FC 82
TITLE = Sheet 5 (ATC)
//LADDERS 3, 5, 9, 600, P00M01-M11 (Digital)
AUTHOR : RJ
FAMILY : ATC
VERSION : 0.1
BEGIN
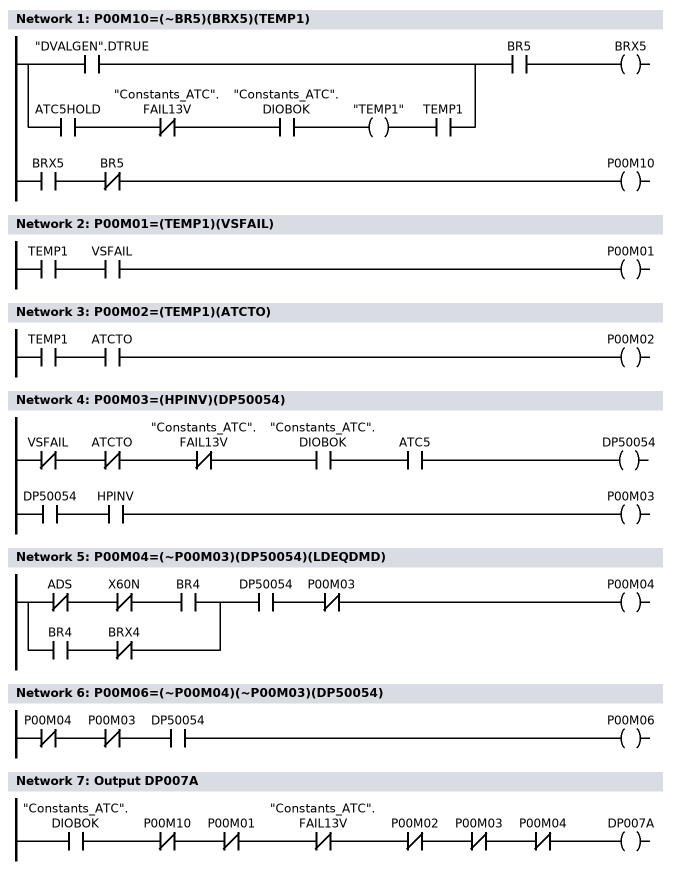
NETWORK
TITLE = P00M10=(~BR5)(BRX5)(TEMP1)
//BRX5=BR5
//TEMP1=(ATC5HOLD)(~FAIL13V)(DIOBOK)
      A(;
      O     "DVALGEN".DTRUE;
      O(;
      A     "ATC5HOLD";
      AN    "Constants_ATC".FAIL13V;
      A     "Constants_ATC".DIOBOK;
      =     "TEMP1";
      A     "TEMP1";
      );
      );
      A     "BR5";
      =     "BRX5";
      A     "BRX5";
      AN    "BR5";
      =     "P00M10";
NETWORK
TITLE = P00M01=(TEMP1)(VSFAIL)
      A     "TEMP1";
      A     "VSFAIL";
      =     "P00M01";
NETWORK
TITLE = P00M02=(TEMP1)(ATCTO)
      A     "TEMP1";
      A     "ATCTO";
      =     "P00M02";
NETWORK
TITLE = P00M03=(HPINV)(DP50054)
//DP50054=(~VSFAIL)(~ATCTO)(~FAIL13V)(DIOBOK)(ATC5)
      AN    "VSFAIL";
      AN    "ATCTO";
      AN    "Constants_ATC".FAIL13V;
      A     "Constants_ATC".DIOBOK;
      A     "ATC5";
      =     "DP50054";
      A     "DP50054";
      A     "HPINV";
      =     "P00M03";
NETWORK
TITLE = P00M04=(~P00M03)(DP50054)(LDEQDMD)
//LDEQDMD=[(~ADS)(~X60N)(BR4)]+[(BR4)(~BRX4)]
      A(;
      AN    "ADS";
      AN    "X60N";
      A     "BR4";
      O;
      A     "BR4";
      AN    "BRX4";
      );
      A     "DP50054";
      AN    "P00M03";
      =     "P00M04";
NETWORK
TITLE = P00M06=(~P00M04)(~P00M03)(DP50054)
      AN    "P00M04";
      AN    "P00M03";
      A     "DP50054";
      =     "P00M06";
NETWORK
TITLE = Output DP007A
//DP007A=DIOBOK+(~P00M10)+(~P00M01)+(~FAIL13V)+(~P00M02)+(~P00M03)+(~P00M04)
      A     "Constants_ATC".DIOBOK;
      AN    "P00M10";
      AN    "P00M01";
      AN    "Constants_ATC".FAIL13V;
      AN    "P00M02";
      AN    "P00M03";
      AN    "P00M04";
      =     "DP007A";
END_FUNCTION

FUNCTION "Sheet 6 (ATC)" : VOID	// FC 83
TITLE = Sheet 6 (ATC)
//LADDERS 7, 9, 13, ATC PERMISSIVE (Digital)
AUTHOR : RJ
FAMILY : ATC
VERSION : 0.1
BEGIN
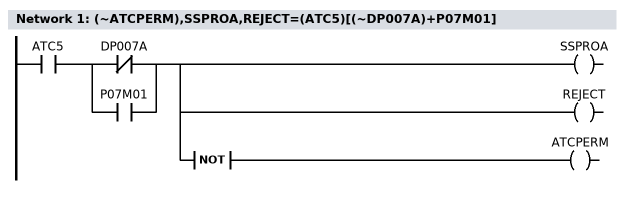
NETWORK
TITLE = (~ATCPERM),SSPROA,REJECT=(ATC5)[(~DP007A)+P07M01]
      A     "ATC5";
      A(;
      ON    "DP007A";
      O     "P07M01";
      );
      =     L 0.0;
      A     L 0.0;
      BLD   102;
      =     "SSPROA";
      A     L 0.0;
      BLD   102;
      =     "REJECT";
      A     L 0.0;
      NOT;
      =     "ATCPERM";
END_FUNCTION

FUNCTION "Sheet 7 (ATC)" : VOID	// FC 84
TITLE = Sheet 7 (ATC)
//LADDER 81. LOOPS 27, 33. WATER COOLED GENERATOR (Analog)
AUTHOR : RJ
FAMILY : ATC
VERSION : 0.1
BEGIN
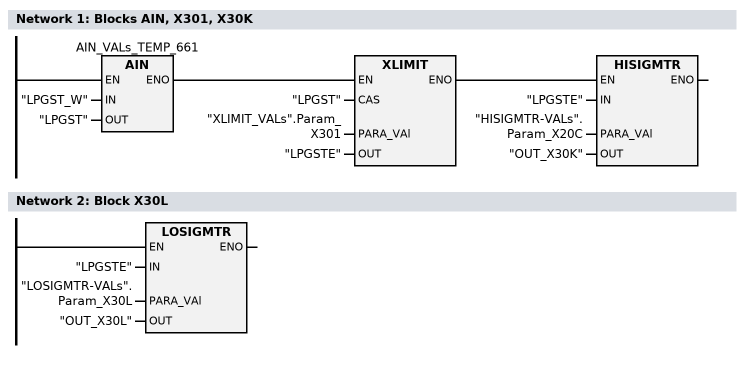
NETWORK
TITLE = Blocks AIN, X301, X30K
      A(;
      A(;
      CALL  "AIN" , "AIN_VALs_TEMP_661" (
           IN                       := "LPGST_W",
           OUT                      := "LPGST");
      A     BR;
      );
      JNB   _001;
      CALL  "XLIMIT" (
           CAS                      := "LPGST",
           PARA_VAl                 := "XLIMIT_VALs".Param_X301,
           OUT                      := "LPGSTE");
_001: A     BR;
      );
      JNB   _002;
      CALL  "HISIGMTR" (
           IN                       := "LPGSTE",
           PARA_VAl                 := "HISIGMTR-VALs".Param_X20C,
           OUT                      := "OUT_X30K");
_002: NOP   0;
NETWORK
TITLE = Block X30L
      CALL  "LOSIGMTR" (
           IN                       := "LPGSTE",
           PARA_VAl                 := "LOSIGMTR-VALs".Param_X30L,
           OUT                      := "OUT_X30L");
      NOP   0;
END_FUNCTION

FUNCTION "Sheet 8 (ATC)" : VOID	// FC 85
TITLE = Sheet 8 (ATC)
//LADDERS 91, 108, 133, GENERATOR ANNUNCIATOR (Digital)
AUTHOR : RJ
FAMILY : ATC
VERSION : 0.1
BEGIN
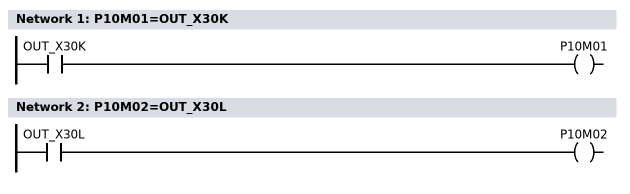
NETWORK
TITLE = P10M01=OUT_X30K
      A     "OUT_X30K";
      =     "P10M01";
NETWORK
TITLE = P10M02=OUT_X30L
      A     "OUT_X30L";
      =     "P10M02";
END_FUNCTION

FUNCTION "Sheet 9 (ATC)" : VOID	// FC 86
TITLE = Sheet 9 (ATC)
//LADDERS 81,83,85,87,109,130. LOOPS 28-30. EXMON & COOLGSHI & P09MXX  (Digital)
AUTHOR : RJ
FAMILY : ATC
VERSION : 0.1
BEGIN
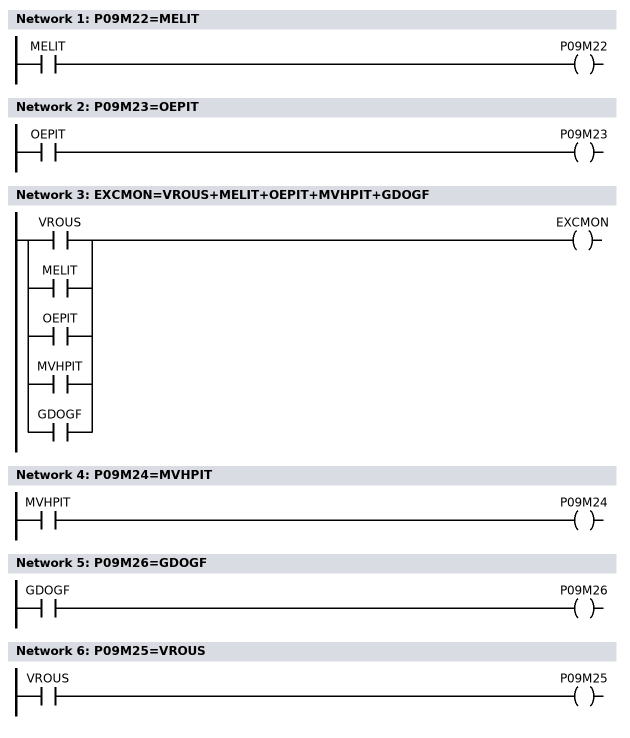
NETWORK
TITLE = P09M22=MELIT
      A     "MELIT";
      =     "P09M22";
NETWORK
TITLE = P09M23=OEPIT
      A     "OEPIT";
      =     "P09M23";
NETWORK
TITLE = EXCMON=VROUS+MELIT+OEPIT+MVHPIT+GDOGF
      O     "VROUS";
      O     "MELIT";
      O     "OEPIT";
      O     "MVHPIT";
      O     "GDOGF";
      =     "EXCMON";
NETWORK
TITLE = P09M24=MVHPIT
      A     "MVHPIT";
      =     "P09M24";
NETWORK
TITLE = P09M26=GDOGF
      A     "GDOGF";
      =     "P09M26";
NETWORK
TITLE = P09M25=VROUS
      A     "VROUS";
      =     "P09M25";
END_FUNCTION

FUNCTION "Sheet 10 (ATC)" : VOID	// FC 87
TITLE = Sheet 10 (ATC)
//LADDERS 31, 34, 36, GENERATOR CALCULATIONS (Analog)
AUTHOR : RJ
FAMILY : ATC
VERSION : 0.1
BEGIN
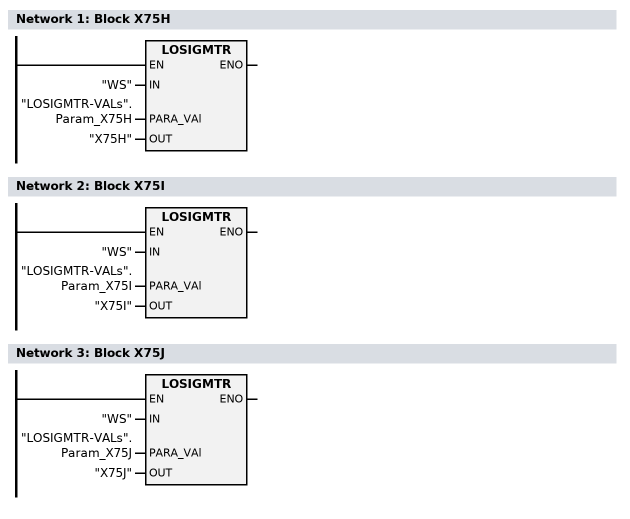
NETWORK
TITLE = Block X75H
      CALL  "LOSIGMTR" (
           IN                       := "WS",
           PARA_VAl                 := "LOSIGMTR-VALs".Param_X75H,
           OUT                      := "X75H");
      NOP   0;
NETWORK
TITLE = Block X75I
      CALL  "LOSIGMTR" (
           IN                       := "WS",
           PARA_VAl                 := "LOSIGMTR-VALs".Param_X75I,
           OUT                      := "X75I");
      NOP   0;
NETWORK
TITLE = Block X75J
      CALL  "LOSIGMTR" (
           IN                       := "WS",
           PARA_VAl                 := "LOSIGMTR-VALs".Param_X75J,
           OUT                      := "X75J");
      NOP   0;
END_FUNCTION

FUNCTION "Sheet 11 (ATC)" : VOID	// FC 88
TITLE = Sheet 11 (ATC)
//LADDERS 15, 17, 18. LOOPS 2, 3. STEAM CHEST - OIL COOLER MONITOR (Analog)
AUTHOR : RJ
FAMILY : ATC
VERSION : 0.1
BEGIN
